PROGRAM MAIN
VAR
	//vnt 1
	bTest_1: BOOL;
	//CNT 2
	bTest_2: BOOL;
END_VAR

END_PROGRAM

(* stored: Version 1.1.0.1, ProductVersion 3.1.4024.12
   POU MAIN: Id {2c2cd341-53ff-4a1d-8582-8b3c7243878f}, SpecialFunc None *)
